// TwinCAT 3 PLC project Reichinger_Katsdorf
// ProgramVersion: 3.1.4023.0
// libraries:
//   EfficientIO Communicator, * (EfficientIO)
//   Lynus Energy Basic, * (Lynus AG)
//   Lynus Energy ModbusTCP, * (Lynus AG)
//   Lynus Persistent Data V1, * (Lynus AG)
//   Lynus Standards, * (Lynus AG)
//   Tc2_ModbusSrv, * (Beckhoff Automation GmbH)
//   Tc2_Standard, * (Beckhoff Automation GmbH)
//   Tc2_System, * (Beckhoff Automation GmbH)
//   Tc2_TcpIp, * (Beckhoff Automation GmbH)
//   Tc2_Utilities, * (Beckhoff Automation GmbH)
//   Tc3_IotBase, * (Beckhoff Automation GmbH)
//   Tc3_Module, * (Beckhoff Automation GmbH)
// project tree:
//   DUTs/ struct_ADS_Reichinger.TcDUT
//   / FastTask.TcTTO, PlcTask.TcTTO, SlowTask.TcTTO
//   FB/ FB_ECS_Alpitronic_Hypercharger_1.TcPOU, FB_EnergyCounter_T.TcPOU, FB_IntervalBit.TcPOU (not stored)
//   POUs/ prgBattery.TcPOU, prgCS.TcPOU, prgEMS.TcPOU, prgGrid.TcPOU, prgHouse.TcPOU, prgLynusCom.TcPOU, prgLynusVar.TcPOU, prgPersistent.TcPOU, prgPV.TcPOU
// real-time tasks:
//   TASK PlcTask: cycle T#10ms, priority 20, ADS port 350
//   TASK SlowTask: cycle T#20ms, priority 21, ADS port 351
//   TASK FastTask: cycle T#5ms, priority 19, ADS port 352

CONFIGURATION Reichinger_Katsdorf
    RESOURCE PLC ON TwinCAT3
        TASK FastTask(INTERVAL := T#5ms, PRIORITY := 19);
        TASK PlcTask(INTERVAL := T#10ms, PRIORITY := 20);
        TASK SlowTask(INTERVAL := T#20ms, PRIORITY := 21);
        PROGRAM prgLynusVar WITH FastTask : prgLynusVar;
        PROGRAM prgPV WITH PlcTask : prgPV;
        PROGRAM prgCS WITH PlcTask : prgCS;
        PROGRAM prgBattery WITH PlcTask : prgBattery;
        PROGRAM prgEMS WITH PlcTask : prgEMS;
        PROGRAM prgPersistent WITH PlcTask : prgPersistent;
        PROGRAM prgGrid WITH PlcTask : prgGrid;
        PROGRAM prgHouse WITH PlcTask : prgHouse;
        PROGRAM prgLynusCom WITH SlowTask : prgLynusCom;
    END_RESOURCE
END_CONFIGURATION

// ---- DUTs/struct_ADS_Reichinger.TcDUT
TYPE struct_ADS_Reichinger :
STRUCT
	int_liveCount		: INT;	
	bIsEnableEMS		: BOOL;
	bStateAllowChrgFromGrid		: BOOL;
	rHeartbeatEMS		: REAL;
	rErrorWarningEMS 	: REAL;
	rReadyEMS 			: REAL;
	iOperationModeEMS 	: INT;
	byMaxDepthOfDischrgEPO 		: BYTE;
	byReserveSOCEPO 	: BYTE;
	byPrioMinChrgBattSOCInEPO 	: BYTE;
	byResChrgfromGridToBatt 	: BYTE;
	uiUpdateTime 		: UINT;
	bEnableEMS			: BOOL;
	rNewBatteryPowerEMS : REAL;
	bHPActivate			: BOOL;
	bAllowChrgFromGrid	: BOOL;
	bControllingState	: BOOL;
	rMainFuseCSEMS		: REAL;
	lrPowerPV_1			: LREAL;
	lrPowerPV_2			: LREAL;
	lrPowerPV_3			: LREAL;
	lrPowerPV_4			: LREAL;
	lrPowerPV_5			: LREAL;
	lrPowerPV_6			: LREAL;
	lrPowerPV_7			: LREAL;
	lrPowerPV_8			: LREAL;
	lrPowerPV_9			: LREAL;
	lrPowerPV_10		: LREAL;
	lrPowerPV			: LREAL;
	lrPowerGrid			: LREAL;
	rSizeGridConn 		: REAL;
	lrPowerBattery		: LREAL;
	dwSOCBattery		: DWORD;
	rTargetPowerBattery	: REAL;
	bIsEnabledBattery	: BOOL;
	bSResetBattery		: BOOL;
	lrActualCapacityBattery		: LREAL;
	lrMaxCapacityBattery 		: LREAL;
	byPrioBattery		: BYTE;
	bEnableBattery		: BOOL;
	bResetBattery		: BOOL;
	lrPowerHouse		: LREAL;
	bEnableHouse		: BOOL;
	bHouseEnabled		: BOOL;
	byStateMinPowerCS	: BYTE;
	rTargetPowerCS		: REAL;
	bIsEnabledCS		: BOOL;
	byPrioCS			: BYTE;
	bySOC_E_CS			: BYTE;
	bySOC_D_CS			: BYTE;
	rMaxPowerCS			: REAL;
	byMinPowerCS		: BYTE;
	bEnabledCS			: BOOL;
	lrCounterCS			: LREAL;
	lrCounterPV			: LREAL;
	lrCounterGridCons	: LREAL;
	lrCounterGridProd	: LREAL;
	lrCounterBattCons	: LREAL;
	lrCounterBattProd	: LREAL;
	lrPowerCS			: LREAL;
	bCarConnected		: BOOL;
	rChrgTime			: REAL;
	iMessageEMS			: int;	
	
END_STRUCT
END_TYPE

// ---- POUs/prgLynusVar.TcPOU
PROGRAM prgLynusVar
VAR
	fbVarInfo		: FB_VarInfo_V3;
	fbRW1			: FB_ReadWrite_V2;
//	fbRW2			: FB_ReadWrite;
END_VAR

fbVarInfo(
	bReadInfo:= , 
	eTMCFile:= eSelectTMCFile.eDontUseTMCFile, 
	eSavePositionTMCFile:= eSavePositionOnPLC.ePostionHardDisk, 
	udiCounterFoundVariables=> , 
	bError=> , 
	bBusy=> , 
	byProgress=> , 
	udiErrorCodeOut=> , 
	eErrorVarInfo_Out=> , 
	sVarWithError=> );
	


fbRW1(
	eUploadType:=  3, // Change + 5 min Intervall  , 
	bBusy=> , 
	bError=> , 
	udiErrorCodeOut=> , 
	eErrorReadWrite_Out=> );
	
// fbRW2(bBusy=> , bError=> , udiErrorCodeOut=> , eErrorReadWrite_Out=> );

END_PROGRAM

// ---- POUs/prgPV.TcPOU
PROGRAM prgPV
VAR
	fbPV					: FB_Symo_PV_Inverter_FLOAT_1_DM_30_Inverter;
	fbPV_2					: FB_Symo_PV_Inverter_FLOAT_1_DM_30_Inverter;
//	fbPV_3					: FB_Symo_PV_Inverter_FLOAT_1_DM_30_Inverter;
	fbPVInt					: FB_PV_Power;
	fbPVCounter				: FB_EnergyCounter_T;
	lrPowerPV				: LREAL;				//{#lynus.ag#()}
	byErrorWarningPV		: BYTE;					//{#lynus.ag#()}
	lrPowerPV_1				: LREAL;				//{#lynus.ag#()}
	lrPowerPV_2				: LREAL;				//{#lynus.ag#()}
	lrPowerPV_3				: LREAL;				//{#lynus.ag#()}
	lrPowerPV_4				: LREAL;				//{#lynus.ag#()}
	lrPowerPV_5				: LREAL;				//{#lynus.ag#()}
	lrPowerPV_6				: LREAL;				//{#lynus.ag#()}
	lrPowerPV_7				: LREAL;				//{#lynus.ag#()}
	lrPowerPV_8				: LREAL;				//{#lynus.ag#()}
	lrPowerPV_9				: LREAL;				//{#lynus.ag#()}
	lrPowerPV_10			: LREAL;				//{#lynus.ag#()}
	lrPowerPV_11			: LREAL;				//{#lynus.ag#()}
END_VAR
VAR PERSISTENT
	lrCounterPV				: LREAL;				//{#lynus.ag#()}
END_VAR

fbPV.arrUnitID_Inverter[1] := 1;
fbPV.arrUnitID_Inverter[2] := 2;
fbPV.arrUnitID_Inverter[3] := 3;
fbPV.arrUnitID_Inverter[4] := 4;
fbPV.arrUnitID_Inverter[5] := 5;
fbPV.arrUnitID_Inverter[6] := 6;
fbPV.arrUnitID_Inverter[7] := 7;
fbPV.arrUnitID_Inverter[8] := 8;

fbPV(
	bEnable:= TRUE, 
	sIPAdress:= '10.0.0.105', 
	arrUnitID_Inverter:= , 
	arrDataSymo10=> , 
	stDataEMPower_PV=> , 
	stDataEMCounter_PV=> , 
	diNrOfEM_OUT_PV=> );

lrPowerPV_1 := fbPV.arrDataSymo10[1].lrPowerAcInverter;
lrPowerPV_2 := fbPV.arrDataSymo10[2].lrPowerAcInverter;
lrPowerPV_3 := fbPV.arrDataSymo10[3].lrPowerAcInverter;
lrPowerPV_4 := fbPV.arrDataSymo10[4].lrPowerAcInverter;
lrPowerPV_5 := fbPV.arrDataSymo10[5].lrPowerAcInverter;
lrPowerPV_6 := fbPV.arrDataSymo10[6].lrPowerAcInverter;
lrPowerPV_7 := fbPV.arrDataSymo10[7].lrPowerAcInverter;
lrPowerPV_8 := fbPV.arrDataSymo10[8].lrPowerAcInverter;

fbPV_2.arrUnitID_Inverter[1] := 8;
fbPV_2.arrUnitID_Inverter[2] := 9;

fbPV_2(
	bEnable:= TRUE, 
	sIPAdress:= '10.0.0.102', 
	arrUnitID_Inverter:= , 
	arrDataSymo10=> , 
	stDataEMPower_PV=> , 
	stDataEMCounter_PV=> , 
	diNrOfEM_OUT_PV=> );

lrPowerPV_9 := fbPV_2.arrDataSymo10[1].lrPowerAcInverter;
lrPowerPV_10 := fbPV_2.arrDataSymo10[2].lrPowerAcInverter;

//fbPV_3.arrUnitID_Inverter[1] := 1;

(*
fbPV_3(
	bEnable:= TRUE, 
	sIPAdress:= , 
	arrUnitID_Inverter:= , 
	arrDataSymo10=> , 
	stDataEMPower_PV=> , 
	stDataEMCounter_PV=> , 
	diNrOfEM_OUT_PV=> );

lrPowerPV_11 := fbPV_3.arrDataSymo10[1].lrPowerAcInverter;
*)
	
fbPVInt(
	bEnable:= TRUE, 
	bPowerDataInvers:= , 
	diNrOfEM_IN_PV:= fbPV.diNrOfEM_OUT_PV, 
	stDataPv=> , 
	diNrOfPv_OUT=> );
	
lrPowerPV := fbPVInt.stDataPv.lrPower + lrPowerPV_9 + lrPowerPV_10;
	byErrorWarningPV := fbPVInt.stDataPv.byErrorWarning;

// EnergyCounter
fbPVCounter(
	byActiveTariff:= 1, 
	lrPowerInput:= 0 - lrPowerPV, 
	lrTotalCounterEnergy_Production=> );
	
IF fbPVCounter.lrTotalCounterEnergy_Production > lrCounterPV THEN  	
	lrCounterPV := fbPVCounter.lrTotalCounterEnergy_Production;
END_IF

END_PROGRAM

// ---- FB/FB_EnergyCounter_T.TcPOU

FUNCTION_BLOCK FB_EnergyCounter_T
VAR_INPUT
	byActiveTariff						: BYTE;													//Active Tariff
	lrPowerInput						: LREAL;												//Input Power in kW
END_VAR
VAR_OUTPUT PERSISTENT
	lrTotalCounterEnergy_Consumption	: LREAL;												//Total Counter for Energy consumption with unit kWh
	lrTotalCounterEnergy_Production		: LREAL;												//Total Counter for Energy production with unit kWh
	lrCounterEnergyT1_Consumption		: LREAL;												//Total counter for energy Tariff 1 consumption with unit kWh
	lrCounterEnergyT2_Consumption		: LREAL;												//Total counter for energy Tariff 2 consumption with unit kWh
	lrCounterEnergyT1_Production		: LREAL;												//Total counter for energy Tariff 1 production with unit kWh
	lrCounterEnergyT2_Production		: LREAL;												//Total counter for energy Tariff 2 production with unit kWh
END_VAR
VAR
	arrPD								: ARRAY[1..6] OF FB_PersistentData_Number;				//Function to save persistent data
	timSavePD							: TON;													//Timer to save the persistent Data when the Event Based Mode is active
	timNewValue							: TON;													//Timer to copy every second a new power value
	TaskInfo							: GETCURTASKINDEX;										//Function to get the Task Index
	byWorkMode							: BYTE;													//Work Mode for calculation (1 = Production, 2 = Consumption)
	udiCycleTime						: UDINT;												//Cycle Time
	lrCyclesForSecond					: LREAL;												//Needed cycles for 1 Second
	uiCounterConsumption				: UINT;													//Counter for Cycles in Consumption Mode
	uiSecondsConsumption				: UINT;													//Elapses Seconds for Consumption
	rHourConsumption					: REAL;													//Elapsed Hours for Consumption
	uiCounterProduction					: UINT;													//Counter for Cycles in Production Mode
	uiSecondsProduction					: UINT;													//Elapses Seconds for Production
	rHourProduction						: REAL;													//Elapsed Hours for Production
	lrPowerInput_Int					: LREAL;												//Input Power in kW
	lrkW_Consumption_CP					: LREAL;												//Power to compare in Consumption Mode
	lrkW_Production_CP					: LREAL;												//Powet to compare in Production Mode
END_VAR

//Creator : Kai Ebensperger
//Company : Lynus AG
//Date : 16.11.2021
//Version : 1.0.0.0

//This function block can be used to count different Energy Counter
//Positive Values mens comsumption
//Negative Values means production 

(*--------------------------------------------------------------------------Limits-----------------------------------------------------------------------------------*)

byActiveTariff := LIMIT(1,byActiveTariff,2);

(*---------------------------------------------------------------------------Logic-----------------------------------------------------------------------------------*)

//Get Task Index
TaskInfo(index=> );
	//Cycle Time in ms
	IF TwinCAT_SystemInfoVarList._TaskInfo[TaskInfo.index].CycleTime <> 0 THEN
		udiCycleTime := TwinCAT_SystemInfoVarList._TaskInfo[TaskInfo.index].CycleTime / 10000;
	END_IF

//Cycles for 1 Second
IF udiCycleTime > 0 THEN 
	lrCyclesForSecond := (1 / UDINT_TO_LREAL(udiCycleTime)) * 1000; 
END_IF

//Timer to copy the new Value
//Necessary becaue the rest of the logic can handly min every second a change on the power side
timNewValue(IN:= NOT timNewValue.Q, PT:= T#1S, Q=> , ET=> );
	IF timNewValue.Q THEN lrPowerInput_Int := lrPowerInput; END_IF

IF lrCyclesForSecond <> 0 THEN

	uiCounterConsumption := uiCounterConsumption + 1;
		uiCounterProduction := uiCounterProduction + 1;
	
	//Calculate the Time	
	IF uiCounterProduction >= lrCyclesForSecond THEN uiSecondsProduction := uiSecondsProduction + 1; uiCounterProduction := 0; END_IF
		rHourProduction := UINT_TO_REAL(uiSecondsProduction) / 3600;
	IF uiCounterConsumption >= lrCyclesForSecond THEN uiSecondsConsumption := uiSecondsConsumption + 1; uiCounterConsumption := 0; END_IF
		rHourConsumption := UINT_TO_REAL(uiSecondsConsumption) / 3600;
	
	//Production
	IF lrkW_Production_CP <> lrPowerInput_Int THEN
		IF byWorkMode = 1 THEN 
			//Production Tariff 1
			IF byActiveTariff = 1 THEN 
				lrCounterEnergyT1_Production := lrCounterEnergyT1_Production + ((lrkW_Production_CP * - 1) * rHourProduction); 
					lrkW_Production_CP := lrPowerInput_Int;
			END_IF
			//Production Tariff 2
			IF byActiveTariff = 2 THEN 
				lrCounterEnergyT2_Production := lrCounterEnergyT2_Production + ((lrkW_Production_CP * - 1) * rHourProduction); 
					lrkW_Production_CP := lrPowerInput_Int;
			END_IF
		ELSE
			lrkW_Production_CP := 0;
		END_IF
				rHourProduction := 0; uiSecondsProduction := 0;  uiCounterProduction := 0;	
	END_IF
	
	//Consumption
	IF lrkW_Consumption_CP <> lrPowerInput_Int THEN
		IF byWorkMode = 2 THEN  
			//Consumption Tariff 1
			IF byActiveTariff = 1 THEN 
				lrCounterEnergyT1_Consumption := lrCounterEnergyT1_Consumption + (lrkW_Consumption_CP * rHourConsumption); 
					lrkW_Consumption_CP := lrPowerInput_Int;
			END_IF
			//Consumption Tariff 2
			IF byActiveTariff = 2 THEN 
				lrCounterEnergyT2_Consumption := lrCounterEnergyT2_Consumption + (lrkW_Consumption_CP * rHourConsumption); 
					lrkW_Consumption_CP := lrPowerInput_Int;
			END_IF
		ELSE
			lrkW_Consumption_CP := 0;
		END_IF
				rHourConsumption := 0; uiSecondsConsumption := 0;  uiCounterConsumption := 0;	
	END_IF

END_IF

//Total Consumption and Production
lrTotalCounterEnergy_Consumption := lrCounterEnergyT1_Consumption + lrCounterEnergyT2_Consumption;
	lrTotalCounterEnergy_Production := lrCounterEnergyT1_Production + lrCounterEnergyT2_Production;

//Switch between the Work modes
IF lrPowerInput_Int <= 0 THEN byWorkMode := 1; ELSE byWorkMode := 2; END_IF 
	
(*----------------------------------------------------------Save persistent data----------------------------------------------------------------*)

//When the Event Based mode is active, save the Data only every 6h
//When we have this Function Blocks in the plc code use the Mode "Power Fail" if the PLC System has this possibility
timSavePD(IN:= GVL_Persistent_Data.bEventBasedActive AND NOT timSavePD.Q, PT:= T#6H, Q=> , ET=> );

IF timSavePD.Q THEN
	arrPD[1].lrValue := lrTotalCounterEnergy_Consumption;
	arrPD[2].lrValue := lrTotalCounterEnergy_Production;
	arrPD[3].lrValue := lrCounterEnergyT1_Consumption; 
	arrPD[4].lrValue := lrCounterEnergyT2_Consumption;
	arrPD[5].lrValue := lrCounterEnergyT1_Production;
	arrPD[6].lrValue := lrCounterEnergyT2_Production;
END_IF

arrPD[1](lrValue:= , bEventBasedActive=> );
arrPD[2](lrValue:= , bEventBasedActive=> );
arrPD[3](lrValue:= , bEventBasedActive=> );
arrPD[4](lrValue:= , bEventBasedActive=> );
arrPD[5](lrValue:= , bEventBasedActive=> );
arrPD[6](lrValue:= , bEventBasedActive=> );

END_FUNCTION_BLOCK

// ---- POUs/prgCS.TcPOU
PROGRAM prgCS
VAR PERSISTENT
	bEnabledCS				: BOOL:=TRUE;							//{#lynus.ag#()}
	byPrioCS				: BYTE;									//{#lynus.ag#()}
	bySOC_E_CS				: BYTE;									//{#lynus.ag#()}
	bySOC_D_CS				: BYTE;									//{#lynus.ag#()}
	byMinPowerCS			: BYTE;									//{#lynus.ag#()}
	rMaxPowerCS				: REAL;									//{#lynus.ag#()}
	lrCounterCS				: LREAL;								//{#lynus.ag#()}
END_VAR
VAR
	fbCS					: FB_ECS_Alpitronic_Hypercharger_1;
	fbCSCounter				: FB_EnergyCounter;
	bIsEnabledCS			: BOOL;									//{#lynus.ag#()}
	byErrorWarningCS		: BYTE;									//{#lynus.ag#()}
	byStateMinPowerCS		: BYTE;									//{#lynus.ag#()}
	rTargetPowerCS			: REAL;									//{#lynus.ag#()}
	bCarConnected			: BOOL;									//{#lynus.ag#()}
	rChrgTime				: REAL;									//{#lynus.ag#()}
	lrPowerCS				: LREAL;								//{#lynus.ag#()}
END_VAR

fbCS.stSetupECS.byDisableSOC := bySOC_D_CS;
	fbCS.stSetupECS.byEnableSOC := bySOC_E_CS;
		fbCS.stSetupECS.byPriority := byPrioCS;
			fbCS.stSetupECS.rMaxPower := rMaxPowerCS;
				fbCS.stSetupECS.byCSMinPower := byMinPowerCS;

fbCS(
	bEnable:= bEnabledCS, 
	bPowerDataInvers:= , 
	byUnitID:= 1,				//Allways 1 
	diNrOfEMS_IN:= prgEMS.fbEMS.diNrOfEMS_OUT, 
	diNrOfEM_IN_CS:= , 
	sIPAdress:= '10.0.0.103', 
	stSetupECS:= , 
	stDataECS=> , 
	diNrOfECS_OUT=> );

bIsEnabledCS := fbCS.stDataECS.bEnabled;
	byStateMinPowerCS := fbCS.stDataECS.bySCSMinPower;
		rTargetPowerCS := fbCS.stDataECS.rTargetPower;	
			byErrorWarningCS := fbCS.stDataECS.byErrorWarning;
				bCarConnected := fbCS.stDataECS.bCarConnected;
					rChrgTime := fbCS.stDataECS.arrChargingTimeInMin[1];
						lrPowerCS := fbCS.stDataECS.lrTotalPower;
						

// EnergyCounter
fbCSCounter(
	byActiveTariff:= 1, 
	lrPowerInput:= lrPowerCS, 
	lrTotalCounterEnergy_Consumption=> );
	
IF fbCSCounter.lrTotalCounterEnergy_Consumption > lrCounterCS THEN  	
	lrCounterCS := fbCSCounter.lrTotalCounterEnergy_Consumption;
END_IF

END_PROGRAM

// ---- FB/FB_ECS_Alpitronic_Hypercharger_1.TcPOU
FUNCTION_BLOCK FB_ECS_Alpitronic_Hypercharger_1
VAR_INPUT PERSISTENT
	bEnable										: BOOL;																			//{#lynus.ag#()} //Enable the Fuctionblock and his logic
	bPowerDataInvers							: BOOL;																			//With True its possible to invert all received power data from the electric meter
	byElectricFuseLine							: BYTE; 																		//Electric Fuse Line on wich the ECS is connected => 1 2 3 (If 0 then this charging station is not connected to a Electric Fuse Line)
	byUnitID									: BYTE;																			//Unit ID 
	diNrOfEMS_IN								: DINT;																			//Number of EMS what control this Device.
	diNrOfEM_IN_CS								: DINT;																			//Number of the electric meter for incoming power data. (Power Data for this Device)
	sIPAdress									: STRING(15);																	//IP Adress from the Alfen charging station
	stSetupECS									: ST_Setup_ECS;																	//{#lynus.ag#()} //Setup charging station
END_VAR
VAR_OUTPUT
	stDataECS									: ST_ECS_Output;																//{#lynus.ag#()} //Electric charging station output data
	diNrOfECS_OUT								: DINT;																			//Active Number from the Electric charging Function for using on other functions
	lrTotalPowerECSRealTime						: LREAL;																		//Total Electric Power in kW read out directly from the Charging station. (Real time)
END_VAR
VAR
	{attribute 'hide'}
	fbCS										: FB_ElectricChargingStation;													//Function block for electric charging station
	{attribute 'hide'}
	fbNumberDevice								: FB_NumberOfDevice;															//Function block to calcualte the number of the Device
	fbDIExternalLock							: FB_XL1XXX_DI;																	//Digital Input from external loock signal
	{attribute 'hide'}
	fbMBRead_FC4								: FB_MBReadInputRegs ;															//Modbus Read Function (FC4)
	{attribute 'hide'}
	fbMBWrite_FC16								: FB_MBWriteRegs;																//Modbus Write Function (FC16)
	{attribute 'hide'}
	fbConvertDwordToWord						: FB_CV_DWORD_TO_WORD;															//Convert Dword to Word
	{attribute 'hide'}
	fbConvertWordToDord							: FB_CV_WORD_TO_DWORD;															//Convert Word to Dword
	{attribute 'hide'}
	timDelay									: TON;																			//Timer for Delay between Requests
	{attribute 'hide'}
	timTimeout									: TON;																			//Timer for Timeout
	{attribute 'hide'}
	timDissableFunctions						: TON;																			//Timer to dissable the Function after Lynus_Standards.Constants_General.tTimeDissableLynusFunctions Days without connection to the Lynus Cloud
	{attribute 'hide'}
	timResetConnectionOnGVL						: TON;																			//Timer to try reset the connection Flag on the GVL. (When somebody delete the Connection Function and make only a onlinechange)
	{attribute 'hide'}
	timDelayStart								: TON;																			//Timer to start the state machine with Daley after enabling or after the system ist restartet
	{attribute 'hide'}
	FPError_FC_4								: R_TRIG;																		//Internal positive Edge
	{attribute 'hide'}
	FPError_FC_16								: R_TRIG;																		//Internal positive Edge
	{attribute 'hide'}
	FPEnable									: R_TRIG;																		//Internal positive Edge
	{attribute 'hide'}
	arrPD										: ARRAY[1..15] OF FB_PersistentData_Number;										//Function to save persistent data
	{attribute 'conditionalshow'}
	arrEnergyCounterSocket						: ARRAY[1..4] OF FB_EnergyCounter;												//FB energy Counter, because the charging station not deliver the total energy Counter in kWh
	{attribute 'hide'}
	fbPDString									: FB_PersistentData_String;														//Function to save persistent string data
	{attribute 'hide'}
	arrBuffer_FC4								: ARRAY[1..9] OF WORD;															//Buffer with Data from FC3
	{attribute 'hide'}
	arrBuffer_FC16								: ARRAY[1..2] OF WORD;															//Buffer with Data from FC16
	{attribute 'hide'}
	arrConnectorState							: ARRAY[1..4] OF WORD;															//Connector State
	{attribute 'hide'}
	arrChargingTime								: ARRAY[1..4] OF WORD;															//Charging Time in seconds
	{attribute 'hide'}
	arrSOCCar									: ARRAY[1..4] OF WORD;															//SOC from the Car
	{attribute 'hide'}
	arrPowerConnector							: ARRAY[1..4] OF DWORD;															//Power in W from each Connector
	{attribute 'hide'}
	arrEnergySession							: ARRAY[1..4] OF REAL;															//Energy Session in kWh
	{attribute 'hide'}
	bErrorCS									: BOOL;																			//Error State from the charging station
	{attribute 'hide'}
	bMBTCPError									: BOOL;																			//Modbus TCP Function Error																	
	{attribute 'hide'}
	byWaitInStep								: BYTE;																			//Wait in Step before start to clean data on PLC
	{attribute 'hide'}
	iStateGVLData								: INT;																			//State machine to handle the data on the GVL
	{attribute 'hide'}
	iStateModbusRead							: INT;																			//State machine for read out Data over Modbus RTU
	{attribute 'hide'}
	iStateModbusWrite							: INT;																			//State machine for write Data over Modbus RTU
	{attribute 'hide'}
	iStateModbusError							: INT;																			//State machine for error out Data over Modbus RTU	
	{attribute 'hide'}
	iStateModbus_CP								: INT;																			//Variable to compare the state machine variable to set or reset the timeout timer
	{attribute 'hide'}
	wNumberOfConnectors							: WORD;																			//Number of real connecotrs on the charging station
	{attribute 'hide'}
	wStationState								: WORD;																			//Charging Station State
	{attribute 'hide'}
	wConnectorInProgress						: WORD;																			//Shows the Connector in Progress when we have more then 1 Connector	
	{attribute 'hide'}
	diNumberOfActiveBatterys					: DINT;																			//Number of active batterys
	{attribute 'hide'}
	diNumberOfBatteryInverterInEPO				: DINT;																			//Number of battery inverters that work in Emergency Power operation 
	{attribute 'hide'}
	diLPForGVL									: DINT;																			//Loop to clean old data on GVL
	{attribute 'hide'}
	diCounterForGVL								: DINT;																			//Counter to clean old data on GVL
	{attribute 'hide'}
	dwSumSOC									: DWORD;																		//Sum of the SOC from all batterys
	{attribute 'hide'}
	dwTargetPower								: DWORD;																		//Target Power in Watt to send to the charging station
	{attribute 'hide'}
	liLPBatteryData								: LINT;																			//Loop to check some data from batterys
	{attribute 'hide'}
	liLPInEPO									: LINT;																			//Loop to check if 1 or more battery inverters build a island grid
END_VAR
VAR PERSISTENT
	{attribute 'conditionalshow'}
	diNrOfEMS_IN_CP								: DINT;																			//Number of EMS what control this Device to compare with the original
END_VAR

//Creator : Kai Ebensperger
//Company : Lynus AG
//Date : 07.10.2021
//Version : 1.0.0.0

//With this Funcition its possible to communicate with a Alpitronic Hypercharger charging station over Modbus TCP.
//Its possible to controll the charging station over the charge power with the unit W
//This Charging station is a DC Hypercharger System.
//This API deliver the real Number of Connectors on the charging station
//To switch off the charging station send 0 Power to the charging station
//The minimal Curretn is set to 7.5 Ampere on AC site, bacause with al values that are < 5kW its not possible to charge the Car on DC site
//This Function Block support maximal 4 Connectors

//Versions that are supported : 1.3A Date : October 2020

//NOTE for diNr.....Designation => 
//_IN = Here Data come in from other Functions or go out to other functions about the GVL
//_OUT = Here Data go out to other functions about the GVL

(*--------------------------------------------------------------------------------------------Limits-------------------------------------------------------------------------------------*)

diNrOfEMS_IN := LIMIT(0,diNrOfEMS_IN,Constants_Energy.diMaxNumberOfEMS);
	diNrOfEM_IN_CS := LIMIT(0,diNrOfEM_IN_CS,Constants_Energy.diMaxNumberOfElectricMeters);	

(*------------------------------------------------------------------Power Data----------------------------------------------------------------------------*)

//Energy Counter Functions
arrEnergyCounterSocket[1](
	byActiveTariff:= 1, 
	lrPowerInput:= DWORD_TO_REAL(arrPowerConnector[1]) / 1000, 
	lrTotalCounterEnergy_Consumption=> , 
	lrTotalCounterEnergy_Production=> , 
	lrCounterEnergyT1_Consumption=> , 
	lrCounterEnergyT2_Consumption=> , 
	lrCounterEnergyT1_Production=> , 
	lrCounterEnergyT2_Production=> );
	
arrEnergyCounterSocket[2](
	byActiveTariff:= 1, 
	lrPowerInput:= DWORD_TO_REAL(arrPowerConnector[2]) / 1000, 
	lrTotalCounterEnergy_Consumption=> , 
	lrTotalCounterEnergy_Production=> , 
	lrCounterEnergyT1_Consumption=> , 
	lrCounterEnergyT2_Consumption=> , 
	lrCounterEnergyT1_Production=> , 
	lrCounterEnergyT2_Production=> );

arrEnergyCounterSocket[3](
	byActiveTariff:= 1, 
	lrPowerInput:= DWORD_TO_REAL(arrPowerConnector[3]) / 1000, 
	lrTotalCounterEnergy_Consumption=> , 
	lrTotalCounterEnergy_Production=> , 
	lrCounterEnergyT1_Consumption=> , 
	lrCounterEnergyT2_Consumption=> , 
	lrCounterEnergyT1_Production=> , 
	lrCounterEnergyT2_Production=> );	
	
arrEnergyCounterSocket[4](
	byActiveTariff:= 1, 
	lrPowerInput:= DWORD_TO_REAL(arrPowerConnector[4]) / 1000, 
	lrTotalCounterEnergy_Consumption=> , 
	lrTotalCounterEnergy_Production=> , 
	lrCounterEnergyT1_Consumption=> , 
	lrCounterEnergyT2_Consumption=> , 
	lrCounterEnergyT1_Production=> , 
	lrCounterEnergyT2_Production=> );

IF diNrOfEM_IN_CS <> 0 THEN
	//Energy Session Input data
	fbCS.bCalculateEnergySession := FALSE;
	fbCS.arrSocketPowerECS[1] := 0;
	fbCS.arrSocketPowerECS[2] := 0;
	fbCS.arrSocketPowerECS[3] := 0;
	fbCS.arrSocketPowerECS[4] := 0;
	fbCS.arrSocketEnergySession[1] := 0;
	fbCS.arrSocketEnergySession[2] := 0;
	fbCS.arrSocketEnergySession[3] := 0;
	fbCS.arrSocketEnergySession[4] := 0;
		IF NOT bPowerDataInvers THEN
			//Energy meter input data for cs Function block
			fbCS.lrCounterEnergyT1_Consumption := Lynus_Standards.GVL_Energy.stDataElectricMeters[diNrOfEM_IN_CS].lrCounterEnergyT1_Production * 1000;
			fbCS.lrCounterEnergyT2_Consumption := Lynus_Standards.GVL_Energy.stDataElectricMeters[diNrOfEM_IN_CS].lrCounterEnergyT2_Production * 1000;
			fbCS.lrCounterEnergyT1_Production := Lynus_Standards.GVL_Energy.stDataElectricMeters[diNrOfEM_IN_CS].lrCounterEnergyT1_Consumption * 1000;
			fbCS.lrCounterEnergyT2_Production := Lynus_Standards.GVL_Energy.stDataElectricMeters[diNrOfEM_IN_CS].lrCounterEnergyT1_Consumption * 1000;
			fbCS.lrTotalCounterEnergy_Consumption := Lynus_Standards.GVL_Energy.stDataElectricMeters[diNrOfEM_IN_CS].lrTotalCounterEnergy_Production * 1000;
			fbCS.lrTotalCounterEnergy_Production := Lynus_Standards.GVL_Energy.stDataElectricMeters[diNrOfEM_IN_CS].lrTotalCounterEnergy_Consumption * 1000;
				fbCS.lrTotalPowerECS := (Lynus_Standards.GVL_Energy.stDataElectricMeters[diNrOfEM_IN_CS].lrPower * 1000) * - 1;
		ELSE
			//Energy meter input data for cs Function block
			fbCS.lrCounterEnergyT1_Consumption := Lynus_Standards.GVL_Energy.stDataElectricMeters[diNrOfEM_IN_CS].lrCounterEnergyT1_Consumption * 1000;
			fbCS.lrCounterEnergyT2_Consumption := Lynus_Standards.GVL_Energy.stDataElectricMeters[diNrOfEM_IN_CS].lrCounterEnergyT2_Consumption * 1000;
			fbCS.lrCounterEnergyT1_Production := Lynus_Standards.GVL_Energy.stDataElectricMeters[diNrOfEM_IN_CS].lrCounterEnergyT1_Production * 1000;
			fbCS.lrCounterEnergyT2_Production := Lynus_Standards.GVL_Energy.stDataElectricMeters[diNrOfEM_IN_CS].lrCounterEnergyT2_Production * 1000;
			fbCS.lrTotalCounterEnergy_Consumption := Lynus_Standards.GVL_Energy.stDataElectricMeters[diNrOfEM_IN_CS].lrTotalCounterEnergy_Consumption * 1000;
			fbCS.lrTotalCounterEnergy_Production := Lynus_Standards.GVL_Energy.stDataElectricMeters[diNrOfEM_IN_CS].lrTotalCounterEnergy_Production * 1000;
				fbCS.lrTotalPowerECS := Lynus_Standards.GVL_Energy.stDataElectricMeters[diNrOfEM_IN_CS].lrPower * 1000;
		END_IF
ELSE
	//Energy meter input data for cs Function block
	fbCS.lrCounterEnergyT1_Consumption := arrEnergyCounterSocket[1].lrCounterEnergyT1_Consumption + arrEnergyCounterSocket[2].lrCounterEnergyT1_Consumption + arrEnergyCounterSocket[3].lrCounterEnergyT1_Consumption + arrEnergyCounterSocket[4].lrCounterEnergyT1_Consumption;
	fbCS.lrCounterEnergyT1_Consumption := fbCS.lrCounterEnergyT1_Consumption * 1000;
	fbCS.lrCounterEnergyT2_Consumption := arrEnergyCounterSocket[1].lrCounterEnergyT2_Consumption + arrEnergyCounterSocket[2].lrCounterEnergyT2_Consumption + arrEnergyCounterSocket[3].lrCounterEnergyT2_Consumption + arrEnergyCounterSocket[4].lrCounterEnergyT2_Consumption;
	fbCS.lrCounterEnergyT2_Consumption := fbCS.lrCounterEnergyT2_Consumption * 1000;
	fbCS.lrCounterEnergyT1_Production := arrEnergyCounterSocket[1].lrCounterEnergyT1_Production + arrEnergyCounterSocket[2].lrCounterEnergyT1_Production + arrEnergyCounterSocket[3].lrCounterEnergyT1_Production + arrEnergyCounterSocket[4].lrCounterEnergyT1_Production;
	fbCS.lrCounterEnergyT1_Production := fbCS.lrCounterEnergyT1_Production * 1000;
	fbCS.lrCounterEnergyT2_Production := arrEnergyCounterSocket[1].lrCounterEnergyT2_Production + arrEnergyCounterSocket[2].lrCounterEnergyT2_Production + arrEnergyCounterSocket[3].lrCounterEnergyT2_Production + arrEnergyCounterSocket[4].lrCounterEnergyT2_Production;
	fbCS.lrCounterEnergyT2_Production := fbCS.lrCounterEnergyT2_Production * 1000;
	fbCS.lrTotalCounterEnergy_Consumption := fbCS.lrCounterEnergyT1_Consumption + fbCS.lrCounterEnergyT2_Consumption;
	fbCS.lrTotalCounterEnergy_Production := fbCS.lrCounterEnergyT1_Production + fbCS.lrCounterEnergyT2_Production;
		fbCS.lrTotalPowerECS := arrPowerConnector[1] + arrPowerConnector[2] + arrPowerConnector[3] + arrPowerConnector[4];
	//Energy Session Input data
	fbCS.bCalculateEnergySession := FALSE;
	fbCS.arrSocketPowerECS[1] := arrPowerConnector[1];
	fbCS.arrSocketPowerECS[2] := arrPowerConnector[2];
	fbCS.arrSocketPowerECS[3] := arrPowerConnector[3];
	fbCS.arrSocketPowerECS[4] := arrPowerConnector[4];
	fbCS.arrSocketEnergySession[1] := arrEnergySession[1] * 1000;
	fbCS.arrSocketEnergySession[2] := arrEnergySession[2] * 1000;
	fbCS.arrSocketEnergySession[3] := arrEnergySession[3] * 1000;
	fbCS.arrSocketEnergySession[4] := arrEnergySession[4] * 1000;
END_IF			

(*-------------------------------------------------------------Calcualte the number of ECS---------------------------------------------------------------*)

fbNumberDevice(
	diActualNumberOfDevices:= Lynus_Standards.GVL_Energy.stNumberOfDevices.diNumberOfECS, 
	diMaxNumberOfDevices:= Constants_Energy.diMaxNumberOfElectricChargingStations, 
	udiCounterOnlineChange:= TwinCAT_SystemInfoVarList._AppInfo.OnlineChangeCnt, 
	bNumberIsCalculatet=> , 
	bFPNumberIsCalculatet=> , 
	bOnlineChange=> , 
	diNumberForThisDevice=> diNrOfECS_OUT, 
	diNumberOfTotalDevices=> );

//Write new Numer on GVL
IF fbNumberDevice.bFPNumberIsCalculatet THEN
	Lynus_Standards.GVL_Energy.stNumberOfDevices.diNumberOfECS := fbNumberDevice.diNumberOfTotalDevices;	
END_IF 

//Delete old Number on GVL
IF fbNumberDevice.bOnlineChange THEN 
	Lynus_Standards.GVL_Energy.stNumberOfDevices.diNumberOfECS := diNrOfECS_OUT;	
		iStateGVLData := 1;
END_IF

(*-------------------------------------------------------------Service from Backend is ready and check the connection to backen for dissabel/enable Function---------------------------------------------------------------*)

//Try to reset the variable for connection on the GVL. When all is normal then the Lynus Mqtt connection function set this variable to true in the next cycle
//When we have no connection to the backend then after Lynus_Standards.Constants_General.tTimeDissableLynusFunctions days the Function is dissabled with all of his functionalities
timResetConnectionOnGVL(IN:= NOT timResetConnectionOnGVL.Q, PT:= T#1H, Q=> , ET=> );
	IF timResetConnectionOnGVL.Q THEN Lynus_Standards.GVL_Communicator.bStateConnectionToEnableFunctions := FALSE; END_IF
		IF NOT Lynus_Standards.GVL_Communicator.bStateConnectionToEnableFunctions THEN timDissableFunctions.IN := TRUE; ELSE timDissableFunctions.IN := FALSE; END_IF  
			timDissableFunctions(IN:= , PT:= Lynus_Standards.Constants_General.tTimeDissableLynusFunctions, Q=> , ET=> );
			
(*--------------------------------------------------------------------------------------------State Machine Read--------------------------------------------------------------------------------------*)

//Timer for Delay
timDelay(IN:= , PT:= T#250MS, Q=> , ET=> );

//Timer for Timeout in Statemachine
IF (iStateModbusRead > 0 AND iStateModbusRead <= 3 AND iStateModbusRead = iStateModbus_CP) OR
		(iStateModbusWrite > 0 AND iStateModbusWrite <= 1 AND iStateModbusWrite = iStateModbus_CP) THEN
			timTimeout.IN := TRUE;
ELSE	
			timTimeout.IN := FALSE;
END_IF 
	//Timeout Timer is dissabled when the Init Step is aktiv or the function is not enabled
	IF (iStateModbusRead = 0 AND iStateModbusWrite = 0) OR NOT bEnable THEN timTimeout.IN := FALSE; END_IF
		timTimeout(IN:= , PT:= T#10S, Q=> , ET=> );

//Enable with Delay that not all sockets have to be created at the same time
timDelayStart(IN:= bEnable, PT:= T#20MS * diNrOfECS_OUT, Q=> , ET=> );
	FPEnable(CLK:= timDelayStart.Q, Q=> );

IF FPEnable.Q AND iStateModbusRead = 0 AND iStateModbusWrite = 0 THEN iStateModbusRead := 1; wConnectorInProgress := 1; END_IF		
		
//Not Enabled
IF NOT bEnable THEN iStateModbusRead := 0; iStateModbusError := 0; iStateModbusWrite := 0; END_IF		
		
CASE iStateModbusRead OF

	0://Init Step 
		iStateModbus_CP := 0;
			timDelay.IN := FALSE;
				fbMBRead_FC4.bExecute := FALSE;
					fbMBWrite_FC16.bExecute := FALSE;
						wConnectorInProgress := 0;
		arrConnectorState[1] := 0; arrConnectorState[2] := 0; arrConnectorState[3] := 0; arrConnectorState[4] := 0;
	
	1://Read Out the Number of connectors and the Charging station State (Register 2 and 3)
		iStateModbus_CP := iStateModbusRead;
		
		//Reset Write
		fbMBWrite_FC16.bExecute := FALSE;
			
		//Start Read
		fbMBRead_FC4.nQuantity := 2;
			fbMBRead_FC4.nMBAddr := 2;
				fbMBRead_FC4.bExecute := TRUE;
					fbMBRead_FC4.nUnitID := byUnitID;
			
		IF fbMBRead_FC4.bBusy THEN timDelay.IN := TRUE; END_IF
		
		//Wait for Delay, copy Data and then next step
		IF NOT fbMBRead_FC4.bBusy AND NOT fbMBRead_FC4.bError AND timDelay.Q THEN
			//Number of real Connectors
			wNumberOfConnectors := arrBuffer_FC4[1];
			//Charging station State
			wStationState := arrBuffer_FC4[2];	 
			//Connector in Progress
			wConnectorInProgress := LIMIT(1,wConnectorInProgress,4);
			//Go to Next Step
			fbMBRead_FC4.bExecute := FALSE;
				timDelay.IN := FALSE;		
					iStateModbusRead := 2;
		END_IF	

		//Error or Timeout
		IF FPError_FC_4.Q OR timTimeout.Q THEN
			iStateModbusError := 300;
		END_IF
		
	2://Read Out the Information of the real connecotrs (Register "1"00 to "1"08)
		iStateModbus_CP := iStateModbusRead;
		
		//Start Read
		fbMBRead_FC4.nQuantity := 9;
			fbMBRead_FC4.nMBAddr := 100 * wConnectorInProgress;
				fbMBRead_FC4.bExecute := TRUE;
					fbMBRead_FC4.nUnitID := byUnitID;
			
		IF fbMBRead_FC4.bBusy THEN timDelay.IN := TRUE; END_IF
		
		//Wait for Delay, copy Data and then next step
		IF NOT fbMBRead_FC4.bBusy AND NOT fbMBRead_FC4.bError AND timDelay.Q THEN
			//Connecotor State
			arrConnectorState[wConnectorInProgress] := arrBuffer_FC4[1];
			//Connector Power
			fbConvertWordToDord(wInputValue_1:= arrBuffer_FC4[5], wInputValue_2:= arrBuffer_FC4[6], eByteOrderForConvert:= eByteOrder.eBigEndian, dwOutputValue=> );
				arrPowerConnector[wConnectorInProgress] := fbConvertWordToDord.dwOutputValue;
			//Charging Time in Seconds
			arrChargingTime[wConnectorInProgress] := arrBuffer_FC4[7];
			//Energy Session
			arrEnergySession[wConnectorInProgress] := WORD_TO_REAL(arrBuffer_FC4[8]) / 100;
			//SOC from the Car
			arrSOCCar[wConnectorInProgress] := arrBuffer_FC4[9] / 100;
			//Go to Next Step
			fbMBRead_FC4.bExecute := FALSE;
				timDelay.IN := FALSE;		
					iStateModbusRead := 3;
		END_IF	

		//Error or Timeout
		IF FPError_FC_4.Q OR timTimeout.Q THEN
			iStateModbusError := 300;
		END_IF
		
	3://Wait 1 Step to reset the delay counter befor start to write
		iStateModbus_CP := iStateModbusRead;
		
			iStateModbusWrite := 1;
				//-1 because 0 is the Init Step for Read
				iStateModbusRead := - 1;
				
			//Error on Master, changes on Inputs or Timeout
		 	IF timTimeout.Q THEN 
				iStateModbusError := 300; 
					 
			END_IF
	
END_CASE

(*------------------------------------------------------------------Error and Warning----------------------------------------------------------------------------*)	
 
IF wStationState = 10 OR arrConnectorState[1] = 10 OR arrConnectorState[2] = 10 OR arrConnectorState[3] = 10 OR arrConnectorState[4] = 10 THEN bErrorCS := TRUE; ELSE bErrorCS := FALSE; END_IF  

IF timDissableFunctions.Q THEN fbCS.bWarning := TRUE; fbCS.iWarningCode := 0; ELSE fbCS.bWarning := FALSE; END_IF   
	IF Lynus_Standards.GVL_Energy.stNumberOfDevices.diNumberOfECS > Constants_Energy.diMaxNumberOfElectricChargingStations OR bErrorCS OR bMBTCPError THEN 
		fbCS.bError := TRUE;
	ELSE 
		fbCS.bError := FALSE;
			fbCS.iErrorCode := 0;
	END_IF

IF Lynus_Standards.GVL_Energy.stNumberOfDevices.diNumberOfECS > Constants_Energy.diMaxNumberOfElectricChargingStations THEN fbCS.iErrorCode := 1;
ELSIF bErrorCS OR bMBTCPError THEN fbCS.iErrorCode := 0; END_IF

(*------------------------------------------------------------------Logic----------------------------------------------------------------------------*)

//Calcualte the total SOC if we have more then 1 battery in our system
diNumberOfActiveBatterys := 0;
	dwSumSOC := 0;
		FOR liLPBatteryData := 1 TO Constants_Energy.diMaxNumberOfBatterys BY 1 DO
			IF Lynus_Standards.GVL_Energy.stDataOfBatterys[diNrOfEMS_IN,liLPBatteryData].bEnabled THEN diNumberOfActiveBatterys := diNumberOfActiveBatterys + 1; END_IF
				dwSumSOC := dwSumSOC + Lynus_Standards.GVL_Energy.stDataOfBatterys[diNrOfEMS_IN,liLPBatteryData].dwSOC;
		END_FOR
	
IF diNumberOfActiveBatterys > 0 THEN
	fbCS.dwBatterySOC := DINT_TO_DWORD(DWORD_TO_DINT(dwSumSOC) / diNumberOfActiveBatterys);
ELSE
	fbCS.dwBatterySOC := 100;	//When we have no battery in the ems system
END_IF

//Check if one or more Batterysystems or batteryinverter make island mode
diNumberOfBatteryInverterInEPO := 0;
	FOR liLPInEPO := 1 TO Constants_Energy.diMaxNumberOfBatteryInverters BY 1 DO
		IF Lynus_Standards.GVL_Energy.stDataOfBatteryInverters[diNrOfEMS_IN,liLPInEPO].bWorkOnIslandMode THEN fbCS.bEPOIsActive := TRUE; diNumberOfBatteryInverterInEPO := diNumberOfBatteryInverterInEPO + 1; END_IF
	END_FOR 
		IF diNumberOfBatteryInverterInEPO <= 0 THEN fbCS.bEPOIsActive := FALSE; END_IF

//Digital input for external lock signal
fbDIExternalLock(bInvers:= FALSE, bSignal=> );

//Car connected to the ECS  
IF arrConnectorState[1] = 2 OR arrConnectorState[2] = 2 OR arrConnectorState[3] = 2 OR arrConnectorState[4] = 2 OR
	 arrConnectorState[1] = 3 OR arrConnectorState[2] = 3 OR arrConnectorState[3] = 3 OR arrConnectorState[4] = 3 OR 
		arrConnectorState[1] = 6 OR arrConnectorState[2] = 6 OR arrConnectorState[3] = 6 OR arrConnectorState[4] = 6 THEN 
		fbCS.bCarConnected := TRUE; 
ELSE 
		fbCS.bCarConnected := FALSE; 
END_IF 

//Charging time and SOC from the Car
fbCS.arrSocketChargingTimeInput[1] :=  arrChargingTime[1] / 60;
fbCS.arrSocketChargingTimeInput[2] :=  arrChargingTime[2] / 60;
fbCS.arrSocketChargingTimeInput[3] :=  arrChargingTime[3] / 60;
fbCS.arrSocketChargingTimeInput[4] :=  arrChargingTime[4] / 60;

fbCS.arrSOCCar[1] := arrSOCCar[1];
fbCS.arrSOCCar[2] := arrSOCCar[2];
fbCS.arrSOCCar[3] := arrSOCCar[3];
fbCS.arrSOCCar[4] := arrSOCCar[4];

//Mode 3 State
fbCS.arrSocketMode3StateECS[1] := '';
fbCS.arrSocketMode3StateECS[2] := '';
fbCS.arrSocketMode3StateECS[3] := '';
fbCS.arrSocketMode3StateECS[4] := '';
//ECS is Free
IF arrConnectorState[1] = 0 THEN fbCS.arrSocketMode3StateECS[1] := 'A'; END_IF
IF arrConnectorState[2] = 0 THEN fbCS.arrSocketMode3StateECS[2] := 'A'; END_IF
IF arrConnectorState[3] = 0 THEN fbCS.arrSocketMode3StateECS[3] := 'A'; END_IF
IF arrConnectorState[4] = 0 THEN fbCS.arrSocketMode3StateECS[4] := 'A'; END_IF
//ECS Car Connected
IF arrConnectorState[1] = 2 OR arrConnectorState[1] = 6 THEN fbCS.arrSocketMode3StateECS[1] := 'B1'; END_IF
IF arrConnectorState[2] = 2 OR arrConnectorState[2] = 6 THEN fbCS.arrSocketMode3StateECS[2] := 'B1'; END_IF
IF arrConnectorState[3] = 2 OR arrConnectorState[3] = 6 THEN fbCS.arrSocketMode3StateECS[3] := 'B1'; END_IF
IF arrConnectorState[4] = 2 OR arrConnectorState[4] = 6 THEN fbCS.arrSocketMode3StateECS[4] := 'B1'; END_IF
//ECS Car is Charging
IF arrConnectorState[1] = 3 THEN fbCS.arrSocketMode3StateECS[1] := 'C2'; END_IF
IF arrConnectorState[2] = 3 THEN fbCS.arrSocketMode3StateECS[2] := 'C2'; END_IF
IF arrConnectorState[3] = 3 THEN fbCS.arrSocketMode3StateECS[3] := 'C2'; END_IF
IF arrConnectorState[4] = 3 THEN fbCS.arrSocketMode3StateECS[4] := 'C2'; END_IF

//Functionblock ECS
fbCS(
	bEnable:= bEnable AND NOT timDissableFunctions.Q, 
	bError:= ,
	bWarning := ,
	bEPOIsActive:= , 
	bExternalLock:= fbDIExternalLock.bSignal, 
	bCarConnected:= , 
	bWriteWithDelay:= TRUE, 
	bCalculateEnergySession:= ,
	iErrorCode:= , 
	iWarningCode:= , 
	arrSocketChargingTimeInput:= ,
	arrSOCCar:= , 
	dwBatterySOC:= , 
	lrTotalCounterEnergy_Consumption:= , 
	lrTotalCounterEnergy_Production:= , 
	lrCounterEnergyT1_Consumption:= , 
	lrCounterEnergyT2_Consumption:= , 
	lrCounterEnergyT1_Production:= , 
	lrCounterEnergyT2_Production:= , 
	lrTotalPowerECS:= , 
	arrSocketEnergySession:= ,
	rTargetPower:= Lynus_Standards.GVL_Energy.stDataElectricChargingStations[diNrOfEMS_IN,diNrOfECS_OUT].rTargetPowerEMS, 
	rSupplyVoltage:= 692, 
	rMinCurrent:= 7.5, 
	tTimDelayOutput:= T#5S, 
	tDelayError:= T#5S,
	arrSocketMode3StateECS:= ,
	arrSocketPowerECS:= ,
	stSetupECS:= stSetupECS, 
	stDataECSOut=> , 
	stDataECSOutDelay=> stDataECS);

dwTargetPower := REAL_TO_DWORD((stSetupECS.rMaxPower * fbCS.stDataECSOut.rTargetPower) / 100);
	dwTargetPower := dwTargetPower * 1000;

//Real time Power for Output
lrTotalPowerECSRealTime := fbCS.stDataECSOut.lrTotalPower;
	
(*------------------------------------------------------------------------------------------State Machine Write---------------------------------------------------------------------------------------------*)	

CASE iStateModbusWrite OF	

	1://Set the charging power (Reg 0)
		iStateModbus_CP := iStateModbusWrite;
		
			fbMBWrite_FC16.nQuantity := 2;
				fbMBWrite_FC16.nMBAddr := 0;
					fbMBWrite_FC16.bExecute := TRUE;
						fbMBWrite_FC16.nUnitID := byUnitID;
		
		//Prepear the sending Data. Charging Power for the charging station. 
		//Charging power
		fbConvertDwordToWord(dwInputValue:= dwTargetPower, eByteOrderForConvert:= eByteOrder.eBigEndian, wOutputValue_1=> arrBuffer_FC16[1], wOutputValue_2=> arrBuffer_FC16[2]);
		
		IF fbMBWrite_FC16.bBusy THEN timDelay.IN := TRUE; END_IF

		//Wait for Delay and then next step
		IF NOT fbMBWrite_FC16.bBusy AND NOT fbMBWrite_FC16.bError AND timDelay.Q THEN
			fbMBWrite_FC16.bExecute := FALSE;
				timDelay.IN := FALSE;
					bMBTCPError := FALSE; 
						//Restart from new with the Read out part
						iStateModbusRead := 1;
							iStateModbusWrite := 0;
								wConnectorInProgress := wConnectorInProgress + 1;
									IF wConnectorInProgress > 4 OR wConnectorInProgress > wNumberOfConnectors THEN wConnectorInProgress := 1; END_IF
		END_IF
				
		//Error or Timout
		IF FPError_FC_16.Q OR timTimeout.Q THEN
			iStateModbusError := 300;
		END_IF
		
END_CASE	
	
(*------------------------------------------------------------------------------------------State Machine Error---------------------------------------------------------------------------------------------*)	

CASE iStateModbusError OF
	
	300://Error
		iStateModbus_CP := iStateModbusError;
			timDelay.IN := FALSE;
				fbMBRead_FC4.bExecute := FALSE;
					fbMBWrite_FC16.bExecute := FALSE;
						bMBTCPError := TRUE; 		
							//Restart from new with the Read out part after an Error
							iStateModbusRead := 1;	
								iStateModbusError := 0;
									iStateModbusWrite := 0;
						
END_CASE

(*------------------------------------------------------------------------------------------Modbus TCP Functions---------------------------------------------------------------------------------------------*)

fbMBRead_FC4(sIPAddr:= sIPAdress, nTCPPort:= 502,cbLength:= SIZEOF(arrBuffer_FC4), pDestAddr:= ADR(arrBuffer_FC4), tTimeout:= T#10S );
	FPError_FC_4(CLK:= fbMBRead_FC4.bError, Q=> );		

fbMBWrite_FC16(sIPAddr:= sIPAdress, nTCPPort:= 502, cbLength:= SIZEOF(arrBuffer_FC16), pSrcAddr:= ADR(arrBuffer_FC16), tTimeout:= T#10S);	
	FPError_FC_16(CLK:= fbMBWrite_FC16.bError, Q=> );

(*-----------------------------------------------------------Handle data to Global structure for electric charging stations-----------------------------------------------------------------*)

//Delte al old Data on GVL after a online change or change on the variable diNrOfEMS_IDOD
IF diNrOfEMS_IN <> diNrOfEMS_IN_CP AND iStateGVLData = 0 THEN iStateGVLData := 10; END_IF 

CASE iStateGVLData OF
	
	0://Init Step
		byWaitInStep := 0;
			diCounterForGVL := 1;
	
	1://Wait for 4 Steps before clean al Data on GVL
		byWaitInStep := byWaitInStep + 1;
			IF byWaitInStep >= 4 AND fbNumberDevice.bNumberIsCalculatet THEN iStateGVLData := 2; END_IF
				//To much Devices, back to the Init step
				IF byWaitInStep >= 4 AND NOT fbNumberDevice.bNumberIsCalculatet THEN iStateGVLData := 0; END_IF	
			
	2://Clear all Data in GVL
		FOR diLPForGVL := 1 TO Constants_Energy.diMaxNumberOfEMS BY 1 DO 
			Lynus_Standards.GVL_Energy.stDataElectricChargingStations[diLPForGVL,diCounterForGVL].bEnabled := FALSE;
				Lynus_Standards.GVL_Energy.stDataElectricChargingStations[diLPForGVL,diCounterForGVL].bIsControllable := FALSE;
					Lynus_Standards.GVL_Energy.stDataElectricChargingStations[diLPForGVL,diCounterForGVL].byErrorWarning := 0;
						Lynus_Standards.GVL_Energy.stDataElectricChargingStations[diLPForGVL,diCounterForGVL].byPriority := 0;
							Lynus_Standards.GVL_Energy.stDataElectricChargingStations[diLPForGVL,diCounterForGVL].lrPower := 0;
								Lynus_Standards.GVL_Energy.stDataElectricChargingStations[diLPForGVL,diCounterForGVL].lrPowerConsumption := 0;
									Lynus_Standards.GVL_Energy.stDataElectricChargingStations[diLPForGVL,diCounterForGVL].lrPowerProduction := 0;
										Lynus_Standards.GVL_Energy.stDataElectricChargingStations[diLPForGVL,diCounterForGVL].rMaxPower := 0;
											//Set also the target value from ems back here to 0 and not in EMS function because EMS is in Standy when we have a online change (Problem when we delete a ems function and make a online change)
											Lynus_Standards.GVL_Energy.stDataElectricChargingStations[diLPForGVL,diCounterForGVL].rTargetPowerEMS := 0;	
		END_FOR
		
			//Counter for ECS
			diCounterForGVL := diCounterForGVL + 1;
				diCounterForGVL := LIMIT(0,diCounterForGVL,Constants_Energy.diMaxNumberOfElectricChargingStations);
					//Back to the init step
					IF diCounterForGVL >= Constants_Energy.diMaxNumberOfElectricChargingStations THEN iStateGVLData := 0; END_IF

	10://Clear old Data on GVL 		
		Lynus_Standards.GVL_Energy.stDataElectricChargingStations[diNrOfEMS_IN_CP,diNrOfECS_OUT].bEnabled := FALSE;
			Lynus_Standards.GVL_Energy.stDataElectricChargingStations[diNrOfEMS_IN_CP,diNrOfECS_OUT].bIsControllable := FALSE;
				Lynus_Standards.GVL_Energy.stDataElectricChargingStations[diNrOfEMS_IN_CP,diNrOfECS_OUT].byErrorWarning := 0;
					Lynus_Standards.GVL_Energy.stDataElectricChargingStations[diNrOfEMS_IN_CP,diNrOfECS_OUT].byPriority := 0;
						Lynus_Standards.GVL_Energy.stDataElectricChargingStations[diNrOfEMS_IN_CP,diNrOfECS_OUT].lrPower := 0;
							Lynus_Standards.GVL_Energy.stDataElectricChargingStations[diNrOfEMS_IN_CP,diNrOfECS_OUT].lrPowerConsumption := 0;
								Lynus_Standards.GVL_Energy.stDataElectricChargingStations[diNrOfEMS_IN_CP,diNrOfECS_OUT].lrPowerProduction := 0;
									Lynus_Standards.GVL_Energy.stDataElectricChargingStations[diNrOfEMS_IN_CP,diNrOfECS_OUT].rMaxPower := 0;
									
		diNrOfEMS_IN_CP := diNrOfEMS_IN;
			//Back to the init step
			iStateGVLData := 0;

END_CASE 	 

IF diNrOfECS_OUT > 0 AND fbNumberDevice.bNumberIsCalculatet AND diNrOfEMS_IN > 0 THEN
	Lynus_Standards.GVL_Energy.stDataElectricChargingStations[diNrOfEMS_IN,diNrOfECS_OUT].bEnabled := fbCS.stDataECSOut.bEnabled;
		Lynus_Standards.GVL_Energy.stDataElectricChargingStations[diNrOfEMS_IN,diNrOfECS_OUT].bIsControllable := TRUE;
			Lynus_Standards.GVL_Energy.stDataElectricChargingStations[diNrOfEMS_IN,diNrOfECS_OUT].byErrorWarning := fbCS.stDataECSOut.byErrorWarning;
				Lynus_Standards.GVL_Energy.stDataElectricChargingStations[diNrOfEMS_IN,diNrOfECS_OUT].byPriority := fbCS.stDataECSOut.byPriority;
					Lynus_Standards.GVL_Energy.stDataElectricChargingStations[diNrOfEMS_IN,diNrOfECS_OUT].lrPower := fbCS.stDataECSOut.lrTotalPower;
						Lynus_Standards.GVL_Energy.stDataElectricChargingStations[diNrOfEMS_IN,diNrOfECS_OUT].lrPowerConsumption := fbCS.stDataECSOut.lrTotalPowerConsumption;
							Lynus_Standards.GVL_Energy.stDataElectricChargingStations[diNrOfEMS_IN,diNrOfECS_OUT].lrPowerProduction := fbCS.stDataECSOut.lrTotalPowerProduction;
								Lynus_Standards.GVL_Energy.stDataElectricChargingStations[diNrOfEMS_IN,diNrOfECS_OUT].rMaxPower := fbCS.stDataECSOut.rMaxPower;	
END_IF 

(*----------------------------------------------------------Save persistent data----------------------------------------------------------------*)

arrPD[1](lrValue:= BOOL_TO_LREAL(bEnable), bEventBasedActive=> );
arrPD[2](lrValue:= BOOL_TO_LREAL(bPowerDataInvers), bEventBasedActive=> );
arrPD[3](lrValue:= DINT_TO_LREAL(diNrOfEMS_IN), bEventBasedActive=> );
arrPD[4](lrValue:= DINT_TO_LREAL(diNrOfEM_IN_CS), bEventBasedActive=> );
arrPD[5](lrValue:= BOOL_TO_LREAL(stSetupECS.bManualyOn), bEventBasedActive=> );
arrPD[6](lrValue:= BOOL_TO_LREAL(stSetupECS.bOnEmergPowerOff), bEventBasedActive=> );
arrPD[7](lrValue:= BYTE_TO_LREAL(stSetupECS.byCSMinPower), bEventBasedActive=> );
arrPD[8](lrValue:= BYTE_TO_LREAL(stSetupECS.byDisableSOC), bEventBasedActive=> );
arrPD[9](lrValue:= BYTE_TO_LREAL(stSetupECS.byEnableSOC), bEventBasedActive=> );
arrPD[10](lrValue:= BYTE_TO_LREAL(stSetupECS.byManualyTargetPower), bEventBasedActive=> );
arrPD[11](lrValue:= BYTE_TO_LREAL(stSetupECS.byPriority), bEventBasedActive=> );
arrPD[12](lrValue:= REAL_TO_LREAL(stSetupECS.rMaxPower), bEventBasedActive=> );
arrPD[13](lrValue:= DINT_TO_LREAL(diNrOfEMS_IN_CP), bEventBasedActive=> );
arrPD[14](lrValue:= BYTE_TO_LREAL(byUnitID), bEventBasedActive=> );
fbPDString(sText:= sIPAdress, bEventBasedActive=> );

END_FUNCTION_BLOCK

// ---- POUs/prgEMS.TcPOU
PROGRAM prgEMS
VAR PERSISTENT
	byMaxDepthOfDischrgEPO		: BYTE;							//{#lynus.ag#()}
	byPrioMinChrgBattSOCInEPO	: BYTE;							//{#lynus.ag#()}
	byResChrgfromGridToBatt		: BYTE;							//{#lynus.ag#()}
	byReserveSOCEPO				: BYTE;							//{#lynus.ag#()}
	uiUpdateTime				: UINT;							//{#lynus.ag#()}
	bEnableEMS					: BOOL;							//{#lynus.ag#()}
	bAllowChrgFromGrid			: BOOL;							//{#lynus.ag#()}
	rMainFuseCSEMS				: REAL;							//{#lynus.ag#()}
	iOperationModeEMS			: INT;							//{#lynus.ag#()}
END_VAR
VAR
	fbEMS						: FB_EMS;
	bIsEnableEMS				: BOOL;							//{#lynus.ag#()}
	bStateAllowChrgFromGrid		: BOOL;							//{#lynus.ag#()}
	bHPActivate					: BOOL;							//{#lynus.ag#()}
	bControllingState			: BOOL;							//{#lynus.ag#()}
	iMessageEMS					: INT;							//{#lynus.ag#()}
	rHeartbeatEMS				: REAL;							//{#lynus.ag#()}
	rErrorWarningEMS			: REAL;							//{#lynus.ag#()}
	rReadyEMS					: REAL;							//{#lynus.ag#()}
	rNewBatteryPowerEMS			: REAL;							//{#lynus.ag#()}
	fbRestar					: NT_Reboot;
END_VAR

fbEMS.stSetupEMS.bAllowChrgFromGrid := bAllowChrgFromGrid;
	fbEMS.stSetupEMS.byMaxDepthOfDischrgEPO := byMaxDepthOfDischrgEPO;
		fbEMS.stSetupEMS.byPrioMinChrgBattSOCInEPO := byPrioMinChrgBattSOCInEPO;
			fbEMS.stSetupEMS.byResChrgfromGridToBatt := byResChrgfromGridToBatt;
				fbEMS.stSetupEMS.byReserveSOCEPO := byReserveSOCEPO;
					fbEMS.stSetupEMS.rSizeMainFuseCS := rMainFuseCSEMS;
						fbEMS.stSetupEMS.uiUpdateTime := uiUpdateTime;

IF iOperationModeEMS = 0 THEN fbEMS.eOperationMode := E_OperatingMode_EMS.eAllOff;
ELSIF iOperationModeEMS = 1 THEN fbEMS.eOperationMode := E_OperatingMode_EMS.eSelfConsumption;	
ELSIF iOperationModeEMS = 2 THEN fbEMS.eOperationMode := E_OperatingMode_EMS.ePeakLoadCapping;
ELSIF iOperationModeEMS = 3 THEN fbEMS.eOperationMode := E_OperatingMode_EMS.eLoadManagement;			
END_IF

fbEMS(
	bEnable:= bEnableEMS, 
	diNrOfEM_IN_ECS:= , 
	stSetupEMS:= , 
	eOperationMode:= , 
	eSpeedModeBackendController:= E_SpeedModeBackendController_EMS.eSlow, 
	eSpeedModeLocalController:= E_SpeedModeLocalController_EMS.eSlow,
	bActivateHP:= bHPActivate, 
	bControllingState:= TRUE, //bControllingState, 
	rHeartbeat:= rHeartbeatEMS, 
	rErrorWarning:= rErrorWarningEMS, 
	rEnergyOptReady:= rReadyEMS, 
	rNewBattPower:= rNewBatteryPowerEMS, 
	eMessageEMS=> iMessageEMS, 
	bStateEnable=> bIsEnableEMS, 
	bStateAllowChrgFromGrid=> bStateAllowChrgFromGrid, 
	bMissingPowerData=> , 
	bSurplusAvailable=> , 
	byProgress=> , 
	uiState_OUT=> , 
	diNrOfEMS_OUT=> , 
	arrMinPrioReached=> , 
	arrMaxPrioReached=> );
	
fbRestar(
	NETID:= , 
	DELAY:= , 
	START:= , 
	TMOUT:= , 
	BUSY=> , 
	ERR=> , 
	ERRID=> );

END_PROGRAM

// ---- POUs/prgBattery.TcPOU
PROGRAM prgBattery
VAR PERSISTENT
	bEnableBattery				: BOOL;							//{#lynus.ag#()}
	byPrioBattery				: BYTE;							//{#lynus.ag#()}
	lrMaxCapacityBattery		: LREAL;						//{#lynus.ag#()}
	lrCounterBattProd			: LREAL;						//{#lynus.ag#()}
	lrCounterBattCons			: LREAL;						//{#lynus.ag#()}
END_VAR
VAR
	fbBattery					: FB_Xelectrix_Powerbox;
	fbBattCounter				: FB_EnergyCounter;
	bIsEnabledBattery			: BOOL;							//{#lynus.ag#()}
	bResetBattery				: BOOL;							//{#lynus.ag#()}
	bSResetBattery				: BOOL;							//{#lynus.ag#()}
	byErrorWarningBattery		: BYTE;							//{#lynus.ag#()}
	dwSOCBattery				: DWORD;						//{#lynus.ag#()}
	rTargetPowerBattery			: REAL;							//{#lynus.ag#()}
	lrPowerBattery				: LREAL;						//{#lynus.ag#()}
	lrActualCapacityBattery		: LREAL;						//{#lynus.ag#()}
	
	
	rTargetPowerBatt			: REAL;
	lrGrid						: LREAL;
	int_GridState: INT;											//{#lynus.ag#()}
	int_BatteryState: INT;										//{#lynus.ag#()}
	int_OperatingState: INT;									//{#lynus.ag#()}
	int_ErrorState: INT;										//{#lynus.ag#()}

	FB_Interval: FB_IntervalBit;
	m_IslandOperationStart: BOOL;								//{#lynus.ag#()}
	m_IslandOperationOngoing: BOOL;								//{#lynus.ag#()}
	m_IslandOperationStop: BOOL;								//{#lynus.ag#()}
	t_Interval :TIME:=T#30M;
	t_HightTime :TIME:=T#1S;
	
	m_BatteryErrorActive: BOOL;									//{#lynus.ag#()}
	m_BatteryModbusCommError: BOOL;								//{#lynus.ag#()}
	m_BatteryTargetSPError: BOOL;								//{#lynus.ag#()}
	Ton_Delay_BatteryError: Ton;
	Ton_Delay_BatteryModbusError: Ton;
	Ton_Delay_BatterySPError: Ton;
	lrVoltageL1N		: LREAL;								//{#lynus.ag#()}
	lrVoltageL2N		: LREAL;								//{#lynus.ag#()}
	lrVoltageL3N		: LREAL;								//{#lynus.ag#()}
	lrCurrentL1			: LREAL;								//{#lynus.ag#()}
	lrCurrentL2			: LREAL;								//{#lynus.ag#()}
	lrCurrentL3			: LREAL;								//{#lynus.ag#()}
	r_MaxChargePower	: REAL;									//{#lynus.ag#()}
	r_MaxDisChargePower	: REAL;									//{#lynus.ag#()}

END_VAR

fbBattery(
	bEnable:= bEnableBattery, 
	bActivateControl:= TRUE, 
	byUnitID:= 1, 
	byPriority:= byPrioBattery, 
	diNrOfEMS_IN:= prgEMS.fbEMS.diNrOfEMS_OUT, 
	lrMaxCapacityBattery:= lrMaxCapacityBattery, 
	sIPAdress:= '10.0.0.239', 
	bReset:= bResetBattery, 
	stDataXelectrix=> , 
	stDataBatt=> , 
	stDataBattInverter=> , 
	stDataEMPower_Grid=> , 
	stDataEMCounter_Grid=> , 
	diNrOfBatt_OUT=> , 
	diNrOfBattInverter_OUT=> , 
	diNrOfEM_OUT_Grid=> , 
	lrMaxCapacityBattery_OUT=> );
	
//Out
bIsEnabledBattery := fbBattery.stDataBatt.bEnabled;
bSResetBattery := fbBattery.stDataBattInverter.bStateReset;
dwSOCBattery := fbBattery.stDataBatt.dwSOC;
rTargetPowerBattery := fbBattery.stDataBattInverter.rTargetPower;
lrPowerBattery := fbBattery.stDataBatt.lrPower;
lrActualCapacityBattery := fbBattery.lrMaxCapacityBattery_OUT;	
byErrorWarningBattery := fbBattery.stDataBatt.byErrorWarning;
r_MaxChargePower := fbBattery.stDataBattInverter.rMaxChargePower;	
r_MaxDisChargePower := fbBattery.stDataBattInverter.rMaxDisChargePower;						
						
rTargetPowerBatt := Lynus_Standards.GVL_Energy.stDataOfBatteryInverters[1,1].rTargetPowerEMS;
lrGrid := Lynus_Standards.GVL_Energy.stDataGridConnections[1,1].lrPower;


// EnergyCounter
fbBattCounter(
	byActiveTariff:= 1, 
	lrPowerInput:= lrPowerBattery, 
	lrTotalCounterEnergy_Consumption=> , 
	lrTotalCounterEnergy_Production=> );
	
IF fbBattCounter.lrTotalCounterEnergy_Production > lrCounterBattProd THEN  	
	lrCounterBattProd := fbBattCounter.lrTotalCounterEnergy_Production;
END_IF

IF fbBattCounter.lrTotalCounterEnergy_Consumption > lrCounterBattCons THEN  	
	lrCounterBattCons := fbBattCounter.lrTotalCounterEnergy_Consumption;
END_IF


// send e states to cloud
int_GridState 		:= fbBattery.stDataXelectrix.eGridState;
int_BatteryState	:= fbBattery.stDataXelectrix.eBatteryState;
int_OperatingState	:= fbBattery.stDataXelectrix.eOperatingState;
int_ErrorState		:= fbBattery.stDataXelectrix.eErrorState;


// create bits when battery is in island operation

FB_Interval(
	m_Input			:=  prgBattery.fbBattery.stDataXelectrix.eGridState = 2,	//   2 = Island Mode 
	t_Interval 		:= t_Interval , 
	t_HighTime		:= t_HightTime, 
	m_RisingEdge	=> m_IslandOperationStart, 
	m_Interval		=> m_IslandOperationOngoing, 
	m_FallingEdge	=> m_IslandOperationStop);

	
// monitoring Battery status

Ton_Delay_BatteryError (In := fbBattery.stDataXelectrix.eErrorState =2,
						PT :=T#5S,
						Q => m_BatteryErrorActive);

Ton_Delay_BatteryModbusError (	In := fbBattery.stDataXelectrix.eErrorState = 1,
								PT :=T#5M,
								Q => m_BatteryModbusCommError);						

	
Ton_Delay_BatterySPError (	In := ABS((rTargetPowerBattery/100*fbBattery.stDataBattInverter.rMaxChargePower) - lrPowerBattery) > 10 AND fbBattery.stDataXelectrix.eGridState<>2 AND dwSOCBattery < 90,	// not alarming during island operation
							PT :=T#1M,
							Q => m_BatteryTargetSPError);		
							
							
							
// send voltages to cloud
lrVoltageL1N  :=	prgBattery.fbBattery.stDataEMPower_Grid.lrVoltageL1N;
lrVoltageL2N  :=	prgBattery.fbBattery.stDataEMPower_Grid.lrVoltageL2N;
lrVoltageL3N  :=	prgBattery.fbBattery.stDataEMPower_Grid.lrVoltageL3N;
lrCurrentL1	  := 	prgBattery.fbBattery.stDataEMPower_Grid.lrCurrentL1;
lrCurrentL2	  := 	prgBattery.fbBattery.stDataEMPower_Grid.lrCurrentL2;
lrCurrentL3	  := 	prgBattery.fbBattery.stDataEMPower_Grid.lrCurrentL3;

END_PROGRAM

// ---- POUs/prgPersistent.TcPOU
PROGRAM prgPersistent
VAR
	fbUSV		: FB_WritePersistentData_CX81xx;
	
	fb_Reboot		: NT_reboot;
	m_Reboot		: BOOL:=FALSE;
END_VAR

fbUSV(
	eSaveModeData:= eUSVSaveMode.eSaveWhenPowerfail, 
	bLoadPersistentDataOk=> , 
	bPowerFailDetect=> , 
	bError=> , 
	bySaveProcess=> , 
	dwStorageLast24h=> , 
	udiErrorCode=> );
	
fb_Reboot(	netid := '',
			delay := 2,
			start := m_Reboot);

END_PROGRAM

// ---- POUs/prgGrid.TcPOU
PROGRAM prgGrid
VAR PERSISTENT
	rSizeGridConn				: REAL;									//{#lynus.ag#()}
	lrCounterGridProd			: LREAL;								//{#lynus.ag#()}
	lrCounterGridCons			: LREAL;								//{#lynus.ag#()}
END_VAR
VAR
	fbGrid						: FB_Grid_Power;
	lrGridPower					: LREAL;								//{#lynus.ag#()}
	fbGridCounter				: FB_EnergyCounter;
END_VAR

fbGrid(
	bEnable:= TRUE, 
	diNrOfEMS_IN:= prgEMS.fbEMS.diNrOfEMS_OUT, 
	diNrOfEM_IN_Grid:= prgBattery.fbBattery.diNrOfEM_OUT_Grid, 
	rSizeGridConn:= rSizeGridConn, 
	stDataGrid=> , 
	diNrOfGrid_OUT=> );
	
lrGridPower := fbGrid.stDataGrid.lrPower;

// EnergyCounter
fbGridCounter(
	byActiveTariff:= 1, 
	lrPowerInput:= lrGridPower, 
	lrTotalCounterEnergy_Consumption=> , 
	lrTotalCounterEnergy_Production=> );
	
IF fbGridCounter.lrTotalCounterEnergy_Production > lrCounterGridProd THEN  	
	lrCounterGridProd := fbGridCounter.lrTotalCounterEnergy_Production;
END_IF

IF fbGridCounter.lrTotalCounterEnergy_Consumption > lrCounterGridCons THEN  	
	lrCounterGridCons := fbGridCounter.lrTotalCounterEnergy_Consumption;
END_IF

END_PROGRAM

// ---- POUs/prgHouse.TcPOU
PROGRAM prgHouse
VAR
	fbHouse				: FB_HouseC_Power_Virtual;
	bHouseEnabled		: BOOL;						//{#lynus.ag#()}
	lrPowerHouse		: LREAL;					//{#lynus.ag#()}
	lrPowerHouse_temp	: LREAL;					//{#lynus.ag#()}
END_VAR
VAR PERSISTENT
	bEnableHouse		: BOOL;						//{#lynus.ag#()}
END_VAR

fbHouse(
	bEnable:= bEnableHouse, 
	diNrOfEMS_IN:= prgEMS.fbEMS.diNrOfEMS_OUT, 
	bSetDefault:= , 
	lrCounterConsumptionSetDefault:= , 
	lrCounterProductionSetDefault:= , 
	stDataHouseC=> , 
	diNrOfHouseC_OUT=> );
	
bHouseEnabled := fbHouse.stDataHouseC.bEnabled;
// lrPowerHouse := fbHouse.stDataHouseC.lrPower - prgCS.lrPowerCS;	

lrPowerHouse_temp := prgBattery.lrPowerBattery + prgPV.lrPowerPV + prgGrid.lrGridPower - prgCS.lrPowerCS;
lrPowerHouse := max(0,lrPowerHouse_temp);

END_PROGRAM

// ---- POUs/prgLynusCom.TcPOU
PROGRAM prgLynusCom
VAR
	fbCom		: FB_MqttCommunicator_V3;
	
	byte_array : ARRAY[0..1023] OF BYTE;
	struct_transfer	: struct_ADS_Reichinger;
	mSize_to_Big: BOOL;
	uint_size: UINT;
END_VAR

fbCom(
	bConnect:= TRUE, 
	strAuthKey:=  'BMS99299754422' ,	
	sUserName:= '728932ac-dc47-4305-9677-d9533ba4a462', 
	sUserPassword:= 'e135a39e-aace-40b2-aae8-dca1934900e2', 
	eSavePositionCertificate:= eSavePositionOnPLC.ePostionHardDisk, 
	time_HeartBeat_sec := T#15S,	
	bConnected=> , 
	bError=> , 
	hrErrorCode=> , 
	eConnectionState=> , 
	eErrorMessage_Out=> );

(* old
	sUserName:= '4c01ede1-e5b8-4f13-a81d-df39c4a65466', 
	sUserPassword:= 'b3eed962-3618-4324-b46b-0769d46c8328', 
*)



// copy values to struct
struct_transfer.int_liveCount 				:= struct_transfer.int_liveCount+1;
struct_transfer.bIsEnableEMS			  	:= prgEMS.bIsEnableEMS;
struct_transfer.bStateAllowChrgFromGrid		:= prgEMS.bStateAllowChrgFromGrid;
struct_transfer.rHeartbeatEMS				:= prgEMS.rHeartbeatEMS;
struct_transfer.rErrorWarningEMS			:= prgEMS.rErrorWarningEMS;
struct_transfer.rReadyEMS					:= prgEMS.rReadyEMS;
struct_transfer.iOperationModeEMS			:= prgEMS.iOperationModeEMS;
struct_transfer.byMaxDepthOfDischrgEPO		:= prgEMS.byMaxDepthOfDischrgEPO;
struct_transfer.byReserveSOCEPO				:= prgEMS.byReserveSOCEPO;
struct_transfer.byPrioMinChrgBattSOCInEPO	:= prgEMS.byPrioMinChrgBattSOCInEPO;
struct_transfer.byResChrgfromGridToBatt		:= prgEMS.byResChrgfromGridToBatt;
struct_transfer.uiUpdateTime				:= prgEMS.uiUpdateTime;
struct_transfer.bEnableEMS					:= prgEMS.bEnableEMS;
struct_transfer.rNewBatteryPowerEMS			:= prgEMS.rNewBatteryPowerEMS;
struct_transfer.bHPActivate					:= prgEMS.bHPActivate;
struct_transfer.bAllowChrgFromGrid			:= prgEMS.bAllowChrgFromGrid;
struct_transfer.bControllingState			:= prgEMS.bControllingState;
struct_transfer.rMainFuseCSEMS				:= prgEMS.rMainFuseCSEMS;
struct_transfer.lrPowerPV_1					:= prgPV.lrPowerPV_1;
struct_transfer.lrPowerPV_2					:= prgPV.lrPowerPV_2;
struct_transfer.lrPowerPV_3					:= prgPV.lrPowerPV_3;
struct_transfer.lrPowerPV_4					:= prgPV.lrPowerPV_4;
struct_transfer.lrPowerPV_5					:= prgPV.lrPowerPV_5;
struct_transfer.lrPowerPV_6					:= prgPV.lrPowerPV_6;
struct_transfer.lrPowerPV_7					:= prgPV.lrPowerPV_7;
struct_transfer.lrPowerPV_8					:= prgPV.lrPowerPV_8;
struct_transfer.lrPowerPV_9					:= prgPV.lrPowerPV_9;
struct_transfer.lrPowerPV_10				:= prgPV.lrPowerPV_10;
struct_transfer.lrPowerPV					:= prgPV.lrPowerPV;
struct_transfer.lrPowerGrid					:= prgGrid.lrGridPower;
struct_transfer.rSizeGridConn				:= prgGrid.rSizeGridConn;
struct_transfer.lrPowerBattery				:= prgBattery.lrPowerBattery;
struct_transfer.dwSOCBattery				:= prgBattery.dwSOCBattery;
struct_transfer.rTargetPowerBattery			:= prgBattery.rTargetPowerBattery;
struct_transfer.bIsEnabledBattery			:= prgBattery.bIsEnabledBattery;
struct_transfer.bSResetBattery				:= prgBattery.bSResetBattery;
struct_transfer.lrActualCapacityBattery		:= prgBattery.lrActualCapacityBattery;
struct_transfer.lrMaxCapacityBattery		:= prgBattery.lrMaxCapacityBattery;
struct_transfer.byPrioBattery				:= prgBattery.byPrioBattery;
struct_transfer.bEnableBattery				:= prgBattery.bEnableBattery;
struct_transfer.bResetBattery				:= prgBattery.bResetBattery;
struct_transfer.lrPowerHouse				:= prgHouse.lrPowerHouse;
struct_transfer.bEnableHouse				:= prgHouse.bEnableHouse;
struct_transfer.bHouseEnabled				:= prgHouse.bHouseEnabled;

struct_transfer.byStateMinPowerCS			:= prgCS.byStateMinPowerCS;
struct_transfer.rTargetPowerCS				:= prgCS.rTargetPowerCS;
struct_transfer.bIsEnabledCS				:= prgCS.bIsEnabledCS;
struct_transfer.byPrioCS					:= prgCS.byPrioCS;
struct_transfer.bySOC_E_CS					:= prgCS.bySOC_E_CS;
struct_transfer.bySOC_D_CS					:= prgCS.bySOC_D_CS;
struct_transfer.rMaxPowerCS					:= prgCS.rMaxPowerCS;
struct_transfer.byMinPowerCS				:= prgCS.byMinPowerCS;
struct_transfer.bEnabledCS					:= prgCS.bEnabledCS;
struct_transfer.lrCounterCS					:= prgCS.lrCounterCS;
struct_transfer.lrCounterPV					:= prgPV.lrCounterPV;
struct_transfer.lrCounterGridCons			:= prgGrid.lrCounterGridCons;
struct_transfer.lrCounterGridProd			:= prgGrid.lrCounterGridProd;
struct_transfer.lrCounterBattCons			:= prgBattery.lrCounterBattCons;
struct_transfer.lrCounterBattProd			:= prgBattery.lrCounterBattProd;
struct_transfer.lrPowerCS					:= prgCS.lrPowerCS;
struct_transfer.bCarConnected				:= prgCS.bCarConnected;
struct_transfer.rChrgTime					:= prgCS.rChrgTime;
struct_transfer.iMessageEMS					:= prgEMS.iMessageEMS;
(*
struct_transfer.		:= ;
*)


// copy struct to byte array
IF SIZEOF(struct_transfer) > SIZEOF(byte_array) THEN
	memcpy(ADR(byte_array),ADR(struct_transfer),SIZEOF(byte_array));
	uint_size := SIZEOF(struct_transfer);
	mSize_to_Big := TRUE;
ELSE
	memcpy(ADR(byte_array),ADR(struct_transfer),SIZEOF(struct_transfer));
	mSize_to_Big := FALSE;
END_IF
uint_size := SIZEOF(struct_transfer);

END_PROGRAM
